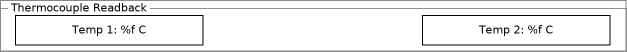
VISUALIZATION VISU_RTDs  // 627x52
VAR_IN_OUT
	fTemp1 : LREAL;
	fTemp2 : LREAL;
END_VAR
    GroupBox (0,0 627x52), "Thermocouple Readback"
        Rectangle (15,15 188x30), "Temp 1: %f C", text variable: fTemp1
        Rectangle (422,15 188x30), "Temp 2: %f C", text variable: fTemp2
END_VISUALIZATION

(* stored: Version 1.1.0.1, ProductVersion 3.1.4024.4
   Visu VISU_RTDs: Id {1b46d21b-55cc-4e7f-ac48-16a84442c307} *)
